(* Schneider Machine Expert - Basic project Proj2, file version 1.6.0.0 *)
(* ProjectInformations: Name=New project *)

HARDWARE
  Cpu 0: TM221CE16R
  EthernetConfiguration: NetworkName=M221, IpAllocationMode=FixedAddress, IpAddress=0.0.0.0, SubnetMask=0.0.0.0
  SerialLineConfiguration: Baud=Baud19200, Parity=ParityEven, DataBits=DataBits8, StopBits=StopBits1, PhysicalMedium=PhysicalMediumRs485, TransmissionMode=TransmissionModeModbusRtu, SlaveId=1, Addressing=SlaveAddressing
  MastTask: UsePeriodScanMode=false, PeriodScan=100
  FastTask: Period=255
  CpuBehavior: StartingMode=StartAsPreviousState, AutoSaveRamOnEeprom=true, WatchdogPeriod=250

SYMBOLS  (address, symbol, comment, settings)

POU New POU
  (* SectionNumber=1 *)

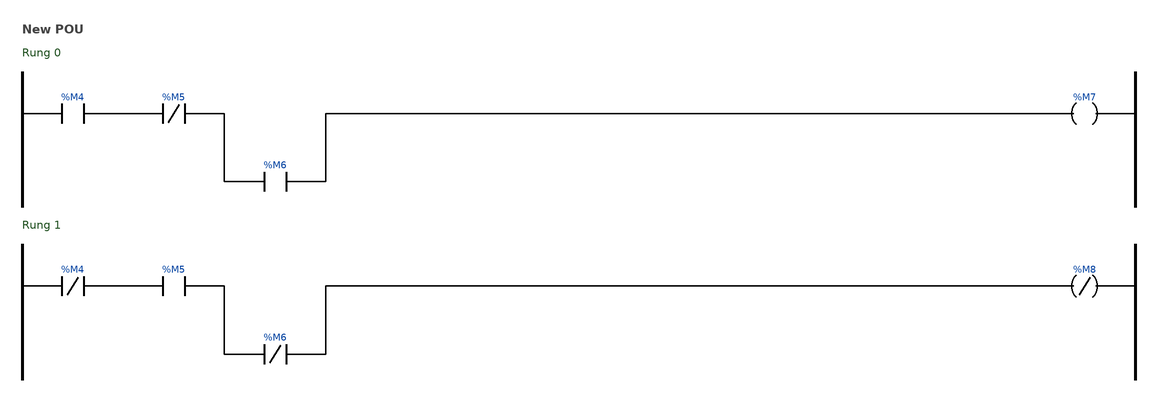

// Rung 0
  LD %M4
  ANDN %M5
  AND %M6
  ST %M7
  // as ST:
  //   %M7 := %M4 AND NOT %M5 AND %M6;

// Rung 1
  LDN %M4
  AND %M5
  ANDN %M6
  STN %M8
  // as ST:
  //   %M8 := NOT (NOT %M4 AND %M5 AND NOT %M6);
